// TIA Portal V20 export
DATA_BLOCK "ET500SP_506"   // DB234
// stored: MemoryReserve 100
   VAR
      "SP506.00 Tab Sensor" : Bool;
      "SP506.01 Tape Sensor" : Bool;
      "SP506.02 VISION TRIGGER SENSOR" : Bool;
      "SP506.03 ELECTRODE PASS KICKER DETECT SENSOR" : Bool;
      "SP506.04 OutputCam_FeedingRollAxisB" : Bool;
      "SP506.05 OutputCam_ElectrodeCutterAxisZ" : Bool;
      "SP506.06 VISION CONTROLLER TRIGGER" : Bool;
      "SP506.07 OutputCam_NgKickerAxisZ" : Bool;
      SPARE1 : Bool;
   END_VAR
BEGIN
END_DATA_BLOCK
